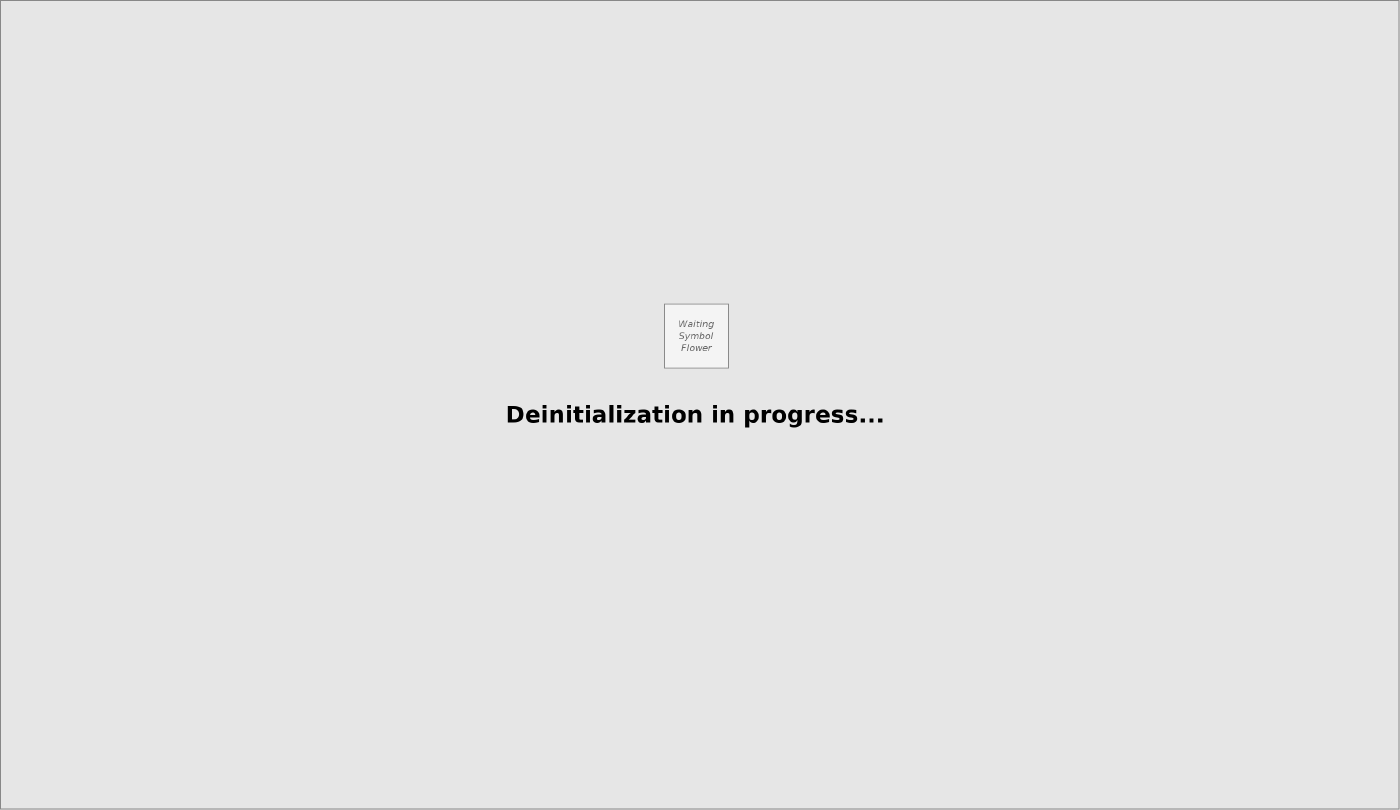
VISUALIZATION PageAborting  // 1520x880
    Group (530,330 450x140)
        WaitingSymbolFlower (191,0 70x70)
        Label (0,100 450x40), "Deinitialization in progress..."
END_VISUALIZATION

// ---- VISUs/Pages/PageAlarms.TcVIS
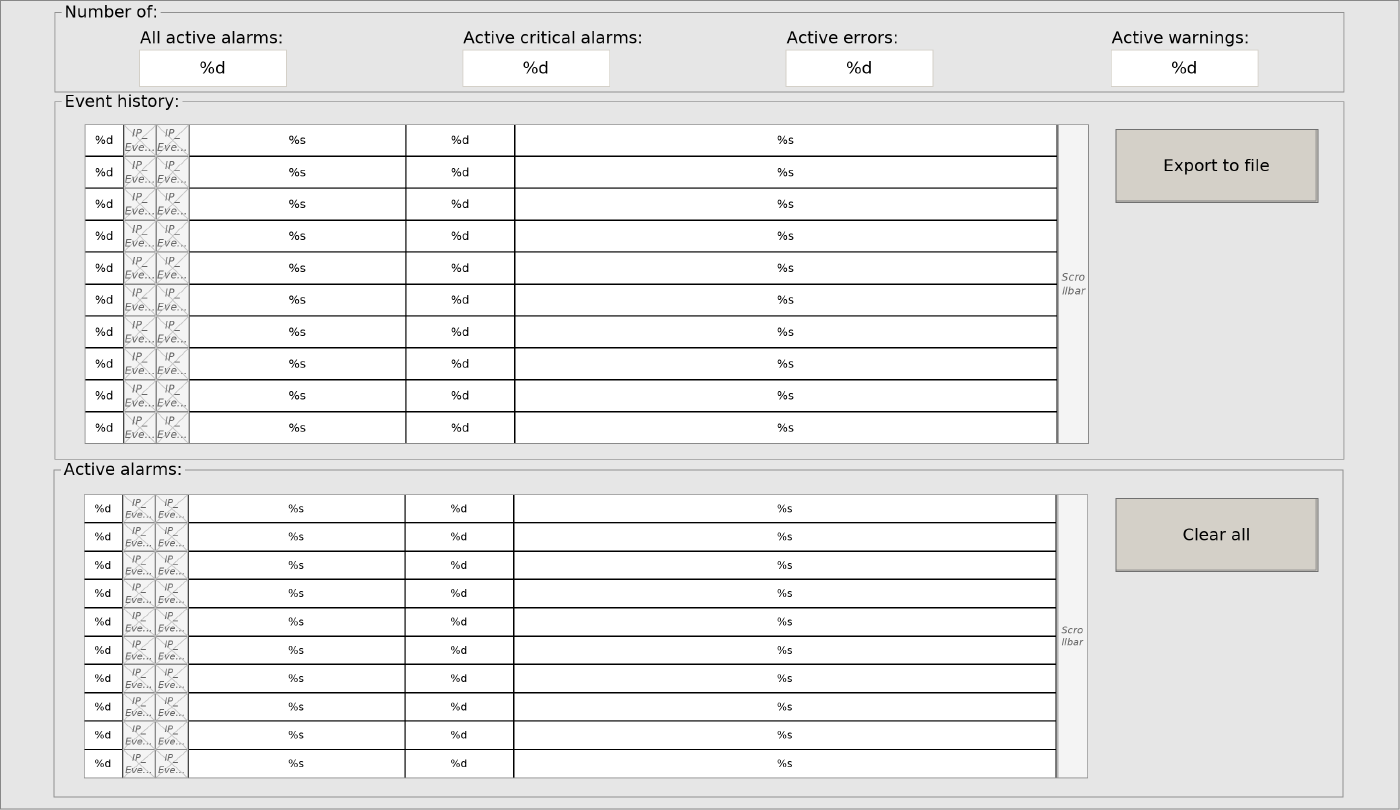
VISUALIZATION PageAlarms  // 1520x880
VAR_IN_OUT
	btnClearAllAlarms 	: BOOL;
	btnExportEvents		: BOOL;
	iActiveAlarms		: UDINT;
	iActiveCritical		: UDINT;
	iActiveErrors		: UDINT;
	iActiveWarrnings	: UDINT;
	arrEvents			: ARRAY[1..PSE_UniversalBlocks.iMAX_EVENTS] OF ST_Event;
	arrAlarms			: ARRAY[1..PSE_UniversalBlocks.iMAX_EVENTS] OF ST_Event;
END_VAR
    GroupBox (58,502 1400x364), "Active alarms:"
        Frame (33,35 1090x308)
            shows EventTable(data := arrAlarms)
        Button (1153,39 220x80), "Clear all"
            tap btnClearAllAlarms
    GroupBox (59,5 1400x95), "Number of:"
        Label (90,21 210x30), "All active alarms:"
        Textfield (92,49 160x40), "%d", text variable: iActiveAlarms, text list: ''
        Label (441,21 234x30), "Active critical alarms:"
        Textfield (443,49 160x40), "%d", text variable: iActiveCritical, text list: ''
        Label (792,21 210x30), "Active errors:"
        Label (1145,21 210x30), "Active warnings:"
        Textfield (794,49 160x40), "%d", text variable: iActiveErrors, text list: ''
        Textfield (1147,49 160x40), "%d", text variable: iActiveWarrnings, text list: ''
    GroupBox (59,102 1400x397), "Event history:"
        Frame (33,33 1090x347)
            shows EventTable(data := arrEvents)
        Button (1152,38 220x80), "Export to file"
            tap btnExportEvents
END_VISUALIZATION

// ---- VISUs/Pages/PageManualCylinders.TcVIS
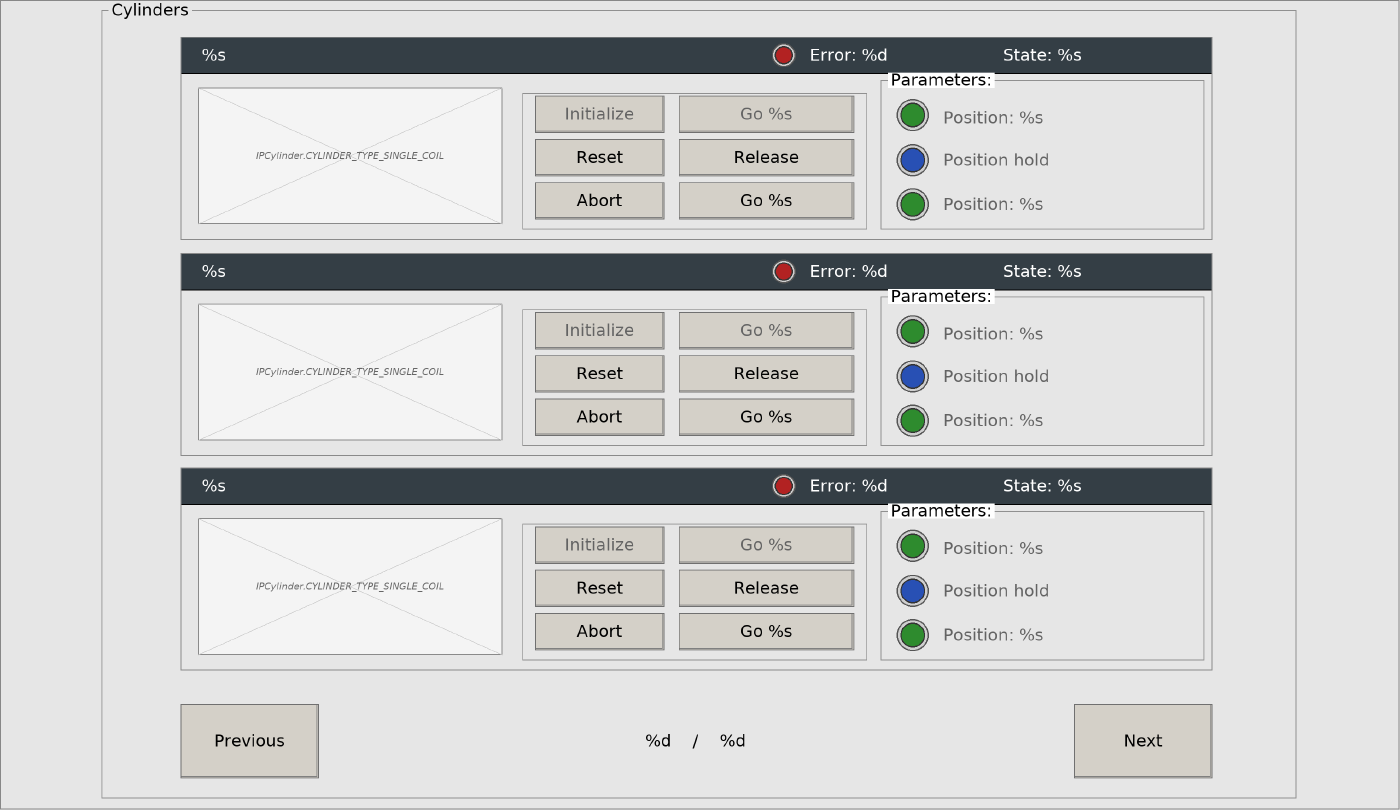
VISUALIZATION PageManualCylinders  // 1520x880
VAR_IN_OUT
	btnPrevious			: BOOL;
	btnNext				: BOOL;
	bPreviousInvisible	: BOOL;
	bNextInvisible		: BOOL;
	stCylinderEmpty		: ARRAY[1..3] OF BOOL;
	stCyliner			: ARRAY[1..3] OF ST_VisuCtrlCylinderFrame;
	iCylinderSelectedPageIndex	: USINT;
	iCylinderTotalPageIndex 	: USINT;
END_VAR
    GroupBox (110,3 1297x864), "Cylinders"
        Button (86,762 150x80), "Previous", invisible if: bPreviousInvisible
            tap btnPrevious
        Button (1056,762 150x80), "Next", invisible if: bNextInvisible
            tap btnNext
        Frame (86,37 1120x220), invisible if: stCylinderEmpty[1]
            shows SingleCylinder(stCylinder := stCyliner[1])
        Frame (86,272 1120x220), invisible if: stCylinderEmpty[2]
            shows SingleCylinder(stCylinder := stCyliner[2])
        Frame (86,505 1120x220), invisible if: stCylinderEmpty[3]
            shows SingleCylinder(stCylinder := stCyliner[3])
        Rectangle (580,777 130x50), "/"
        Rectangle (580,777 50x50), "%d", text variable: iCylinderSelectedPageIndex+1
        Rectangle (661,777 50x50), "%d", text variable: iCylinderTotalPageIndex+1
END_VISUALIZATION

// ---- VISUs/Pages/PageManualRobots.TcVIS
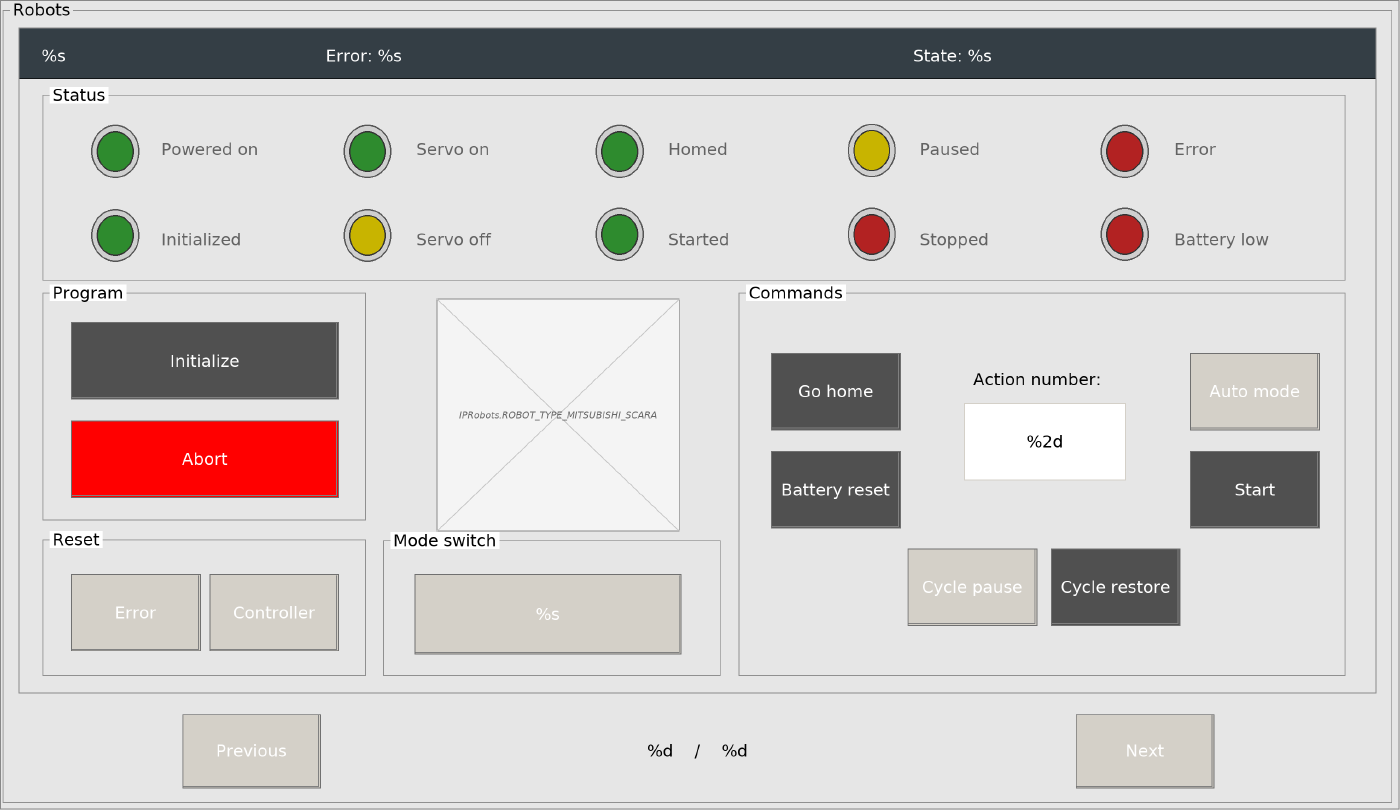
VISUALIZATION PageManualRobots  // 1520x880
VAR_IN_OUT
	btnPrevious			: BOOL;
	btnNext				: BOOL;
	bPreviousInvisible	: BOOL;
	bNextInvisible		: BOOL;
	stRobotEmpty		: ARRAY[1..1] OF BOOL;
	stRobot				: ARRAY[1..1] OF ST_VisuCtrlRobotFrame;
	iRobotSelectedPageIndex	: USINT;
	iRobotTotalPageIndex 	: USINT;
	
END_VAR
    GroupBox (3,3 1508x869), "Robots"
        Button (195,773 150x80), "Previous", invisible if: bPreviousInvisible
            tap btnPrevious
        Button (1165,773 150x80), "Next", invisible if: bNextInvisible
            tap btnNext
        Frame (17,27 1474x723), invisible if: stRobotEmpty[1]
            shows SingleRobot(stRobot := stRobot[1])
        Rectangle (689,788 130x50), "/"
        Rectangle (689,788 50x50), "%d", text variable: iRobotSelectedPageIndex+1
        Rectangle (770,788 50x50), "%d", text variable: iRobotTotalPageIndex+1
END_VISUALIZATION

// ---- VISUs/Pages/PageManualInputs.TcVIS
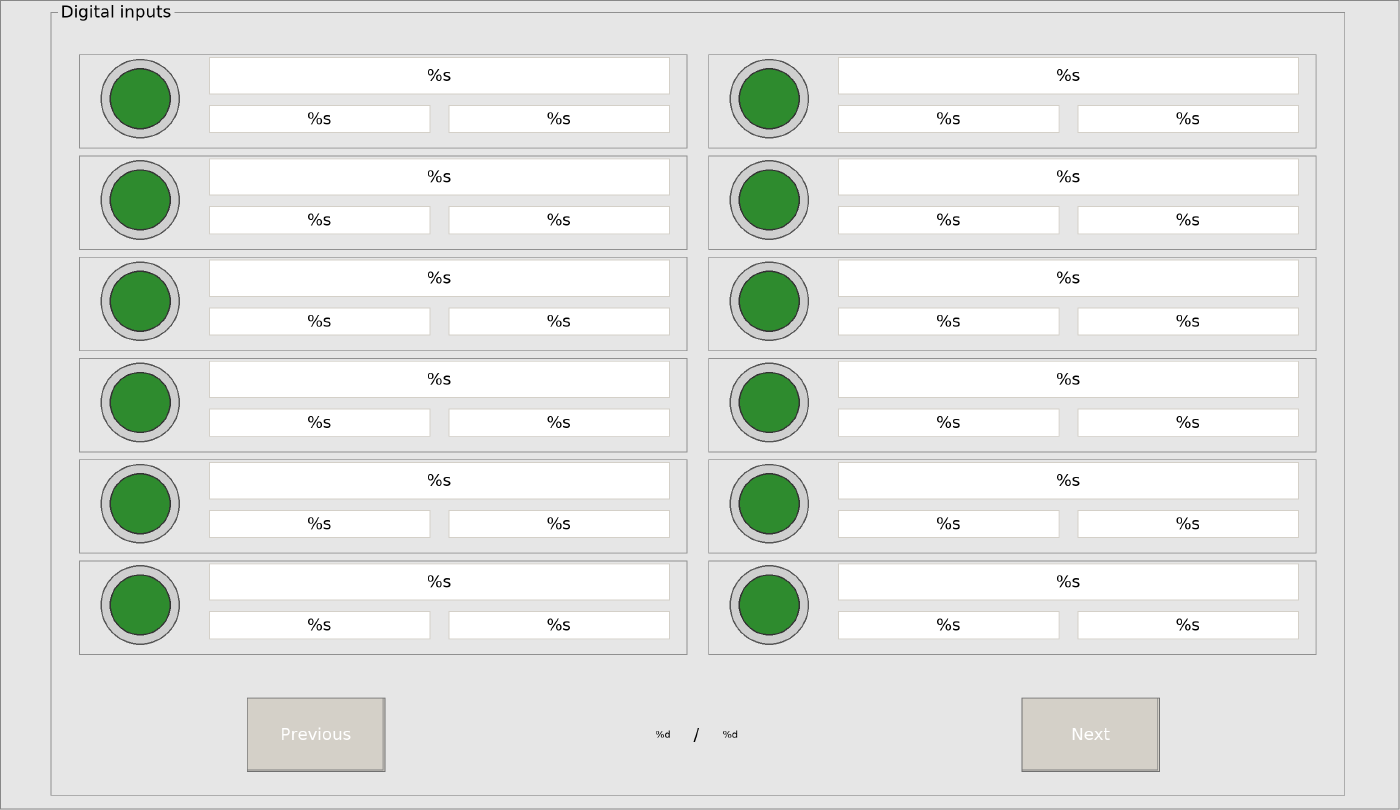
VISUALIZATION PageManualInputs  // 1520x880
VAR_IN_OUT
	btnPrevious			: BOOL;
	btnNext				: BOOL;
	
	bPreviousInvisible	: BOOL;
	bNextInvisible		: BOOL;
	
	stDigitalInputEmpty	: ARRAY[1..12] OF BOOL;
	stDigitalInputData	: ARRAY[1..12] OF ST_VisuCtrlInputFrame;
	
	iInputSelectedPageIndex		: USINT;
	iInputTotalPageIndex 		: USINT;
END_VAR
    GroupBox (55,5 1405x859), "Digital inputs"
        Rectangle (713,768 50x50), "%d", text variable: iInputTotalPageIndex+1
        Rectangle (640,768 50x50), "%d", text variable: iInputSelectedPageIndex+1
        Rectangle (636,768 130x50), "/"
        Button (213,753 150x80), "Previous", invisible if: bPreviousInvisible
            tap btnPrevious
        Button (1054,753 150x80), "Next", invisible if: bNextInvisible
            tap btnNext
        Frame (31,46 660x110), invisible if: stDigitalInputEmpty[1]
            shows SingleDigitalInput(stDigitalInput := stDigitalInputData[1])
        Frame (31,156 660x110), invisible if: stDigitalInputEmpty[2]
            shows SingleDigitalInput(stDigitalInput := stDigitalInputData[2])
        Frame (31,266 660x110), invisible if: stDigitalInputEmpty[3]
            shows SingleDigitalInput(stDigitalInput := stDigitalInputData[3])
        Frame (31,376 660x110), invisible if: stDigitalInputEmpty[4]
            shows SingleDigitalInput(stDigitalInput := stDigitalInputData[4])
        Frame (31,486 660x110), invisible if: stDigitalInputEmpty[5]
            shows SingleDigitalInput(stDigitalInput := stDigitalInputData[5])
        Frame (31,596 660x110), invisible if: stDigitalInputEmpty[6]
            shows SingleDigitalInput(stDigitalInput := stDigitalInputData[6])
        Frame (714,46 660x110), invisible if: stDigitalInputEmpty[7]
            shows SingleDigitalInput(stDigitalInput := stDigitalInputData[7])
    Frame (769,161 660x110), invisible if: stDigitalInputEmpty[8]
        shows SingleDigitalInput(stDigitalInput := stDigitalInputData[8])
    Frame (769,271 660x110), invisible if: stDigitalInputEmpty[9]
        shows SingleDigitalInput(stDigitalInput := stDigitalInputData[9])
    Frame (769,381 660x110), invisible if: stDigitalInputEmpty[10]
        shows SingleDigitalInput(stDigitalInput := stDigitalInputData[10])
    Frame (769,491 660x110), invisible if: stDigitalInputEmpty[11]
        shows SingleDigitalInput(stDigitalInput := stDigitalInputData[11])
    Frame (769,601 660x110), invisible if: stDigitalInputEmpty[12]
        shows SingleDigitalInput(stDigitalInput := stDigitalInputData[12])
END_VISUALIZATION

// ---- VISUs/Pages/PageManualAxis.TcVIS
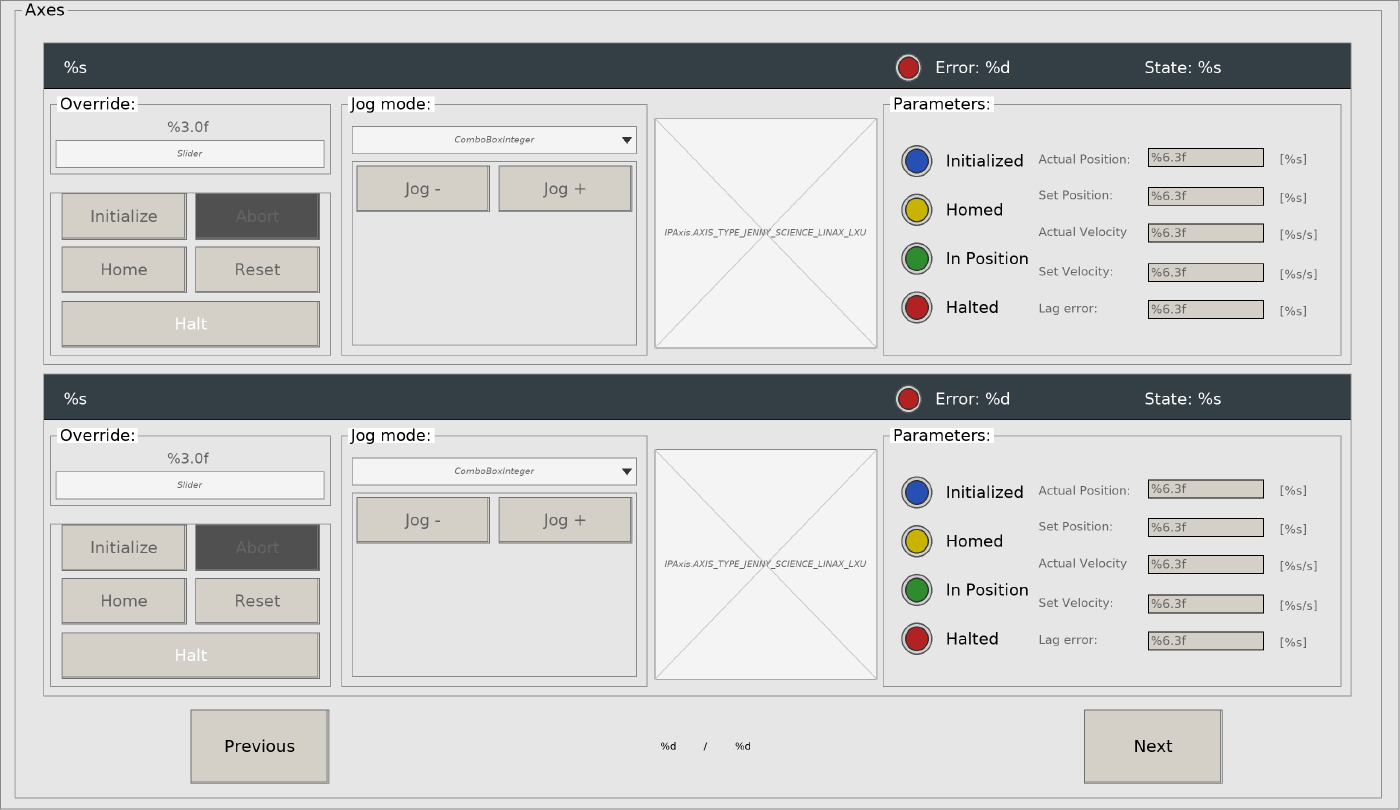
VISUALIZATION PageManualAxis  // 1520x880
VAR_IN_OUT
	btnPrevious			: BOOL;
	btnNext				: BOOL;
	bPreviousInvisible	: BOOL;
	bNextInvisible		: BOOL;
	stAxisEmpty			: ARRAY[0..1] OF BOOL;
	stAxis				: ARRAY[0..1] OF ST_VisuCtrlAxisFrame;
	iAxisSelectedPageIndex		: USINT;
	iAxisTotalPageIndex 		: USINT;
END_VAR
    GroupBox (16,3 1484x864), "Axes"
        Frame (31,43 1420x350), invisible if: stAxisEmpty[0]
            shows SingleAxis(stAxis := stAxis[0])
        Button (1161,768 150x80), "Next", invisible if: bNextInvisible
            tap btnNext
        Button (191,768 150x80), "Previous", invisible if: bPreviousInvisible
            tap btnPrevious
        Frame (31,403 1420x350), invisible if: stAxisEmpty[1]
            shows SingleAxis(stAxis := stAxis[1])
        Rectangle (685,783 130x50), "/"
        Rectangle (685,783 50x50), "%d", text variable: iAxisSelectedPageIndex+1
        Rectangle (766,783 50x50), "%d", text variable: iAxisTotalPageIndex+1
END_VISUALIZATION

// ---- VISUs/Pages/PageManualOutputs.TcVIS
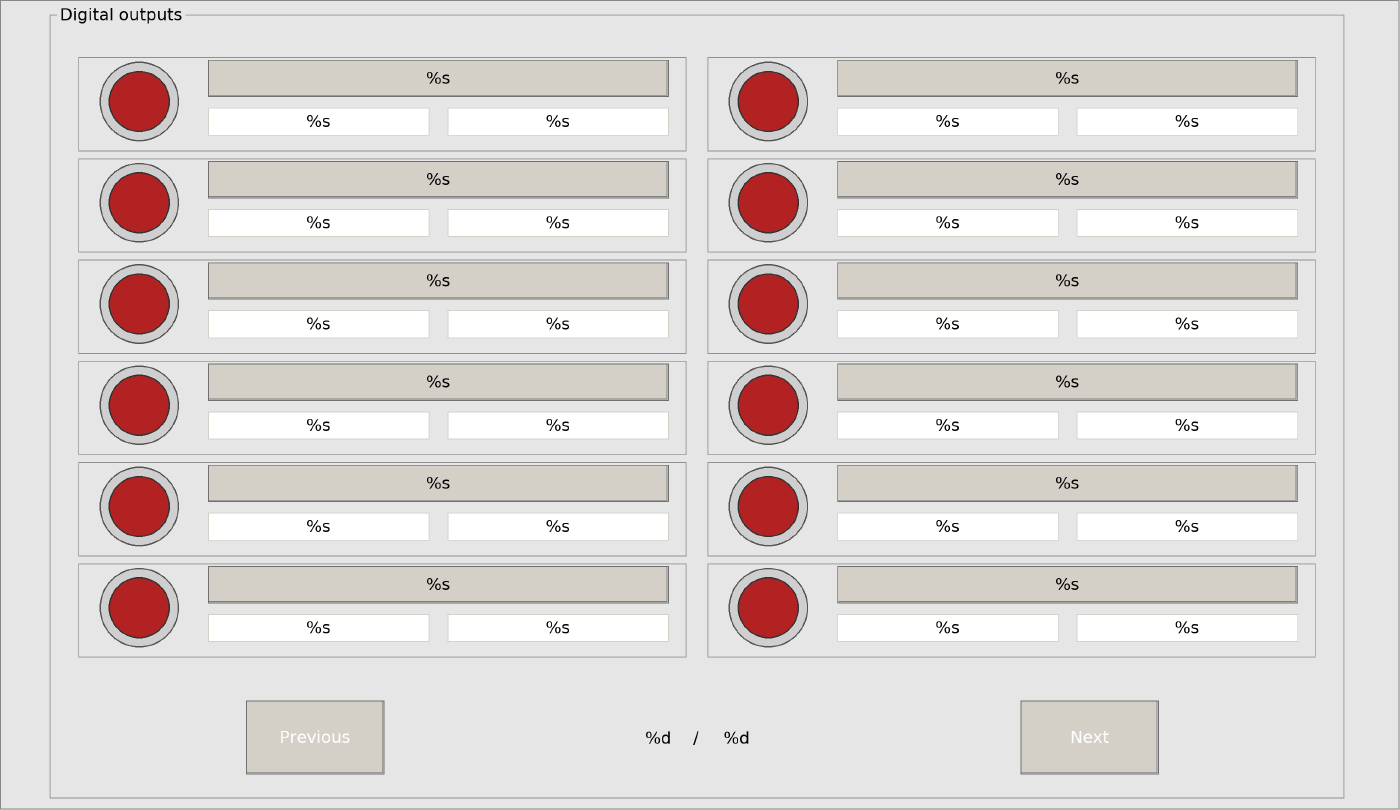
VISUALIZATION PageManualOutputs  // 1520x880
VAR_IN_OUT
	btnPrevious			: BOOL;
	btnNext				: BOOL;
	
	bPreviousInvisible	: BOOL;
	bNextInvisible		: BOOL;
	
	stDigitalOutputEmpty: ARRAY[1..12] OF BOOL;
	stDigitalOutputData	: ARRAY[1..12] OF ST_VisuCtrlOutputFrame;
	
	iOutputSelectedPageIndex	: USINT;
	iOutputTotalPageIndex 		: USINT;
END_VAR
    GroupBox (54,8 1405x859), "Digital outputs"
        Rectangle (721,769 50x50), "%d", text variable: iOutputTotalPageIndex + 1
        Rectangle (636,769 50x50), "%d", text variable: iOutputSelectedPageIndex+1
        Rectangle (636,768 131x51), "/"
        Button (213,753 150x80), "Previous", invisible if: bPreviousInvisible
            tap btnPrevious
        Button (1054,753 150x80), "Next", invisible if: bNextInvisible
            tap btnNext
        Frame (31,46 660x110), invisible if: stDigitalOutputEmpty[1]
            shows SingleDigitalOutput(stDigitalOutput := stDigitalOutputData[1])
        Frame (31,156 660x110), invisible if: stDigitalOutputEmpty[2]
            shows SingleDigitalOutput(stDigitalOutput := stDigitalOutputData[2])
        Frame (31,266 660x110), invisible if: stDigitalOutputEmpty[3]
            shows SingleDigitalOutput(stDigitalOutput := stDigitalOutputData[3])
        Frame (31,376 660x110), invisible if: stDigitalOutputEmpty[4]
            shows SingleDigitalOutput(stDigitalOutput := stDigitalOutputData[4])
        Frame (31,486 660x110), invisible if: stDigitalOutputEmpty[5]
            shows SingleDigitalOutput(stDigitalOutput := stDigitalOutputData[5])
        Frame (31,596 660x110), invisible if: stDigitalOutputEmpty[6]
            shows SingleDigitalOutput(stDigitalOutput := stDigitalOutputData[6])
        Frame (714,46 660x110), invisible if: stDigitalOutputEmpty[7]
            shows SingleDigitalOutput(stDigitalOutput := stDigitalOutputData[7])
    Frame (768,164 660x110), invisible if: stDigitalOutputEmpty[8]
        shows SingleDigitalOutput(stDigitalOutput := stDigitalOutputData[8])
    Frame (768,274 660x110), invisible if: stDigitalOutputEmpty[9]
        shows SingleDigitalOutput(stDigitalOutput := stDigitalOutputData[9])
    Frame (768,384 660x110), invisible if: stDigitalOutputEmpty[10]
        shows SingleDigitalOutput(stDigitalOutput := stDigitalOutputData[10])
    Frame (768,494 660x110), invisible if: stDigitalOutputEmpty[11]
        shows SingleDigitalOutput(stDigitalOutput := stDigitalOutputData[11])
    Frame (768,604 660x110), invisible if: stDigitalOutputEmpty[12]
        shows SingleDigitalOutput(stDigitalOutput := stDigitalOutputData[12])
END_VISUALIZATION

// ---- VISUs/Pages/PageManualSafety.TcVIS
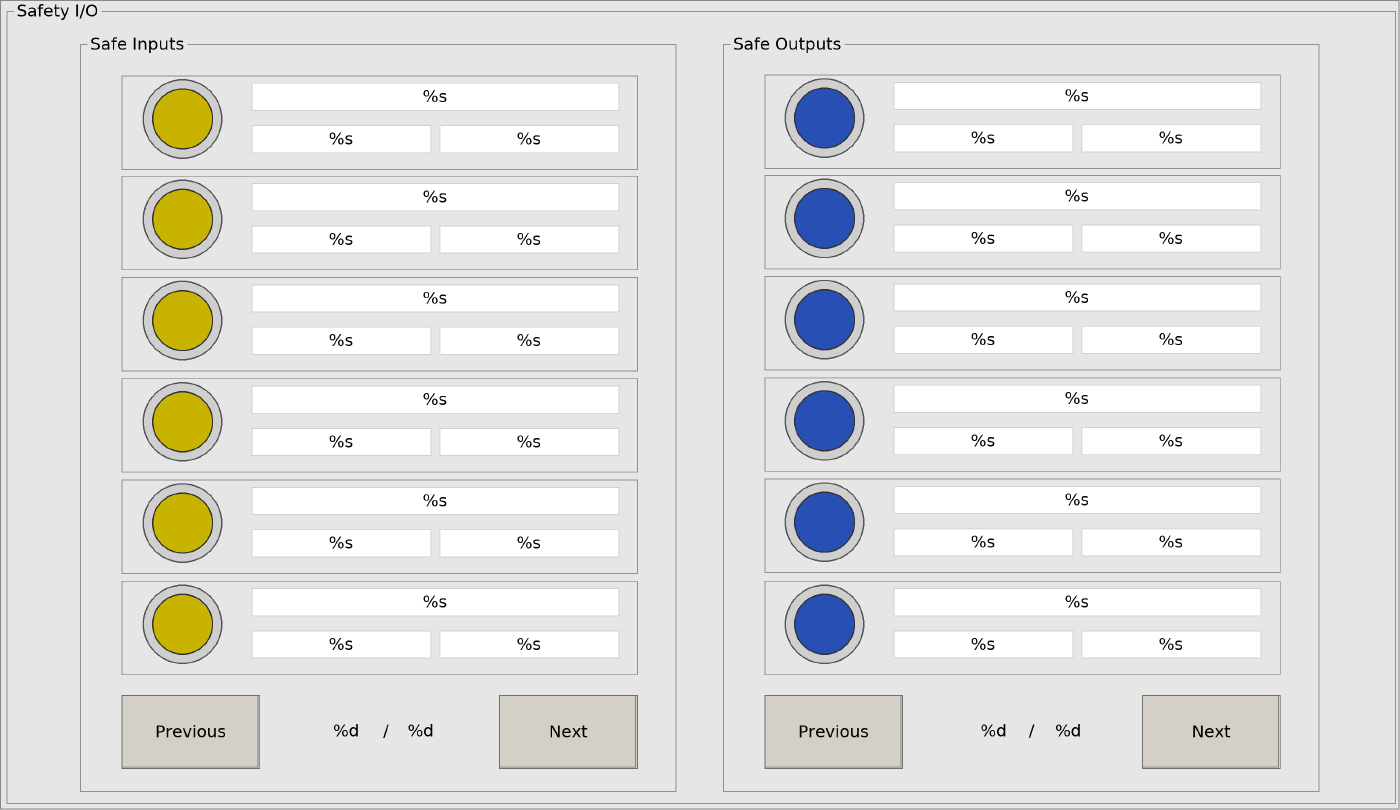
VISUALIZATION PageManualSafety  // 1520x880
VAR_IN_OUT
	btnNextInput			: BOOL;				(*  *)
	btnPreviousInput		: BOOL;				(*  *)
	btnNextOutput			: BOOL;				(*  *)
	btnPreviousOutput		: BOOL;				(*  *)
	
	bNextInvisibleInput		: BOOL;				(*  *)
	bPreviousInvisibleInput	: BOOL;				(*  *)
	bNextInvisibleOutput	: BOOL;				(*  *)
	bPreviousInvisibleOutput: BOOL;				(*  *)	
	
	iSafeInputSelectedPageIndex		: USINT;
	iSafeInputTotalPageIndex 		: USINT;
	iSafeOutputSelectedPageIndex	: USINT;
	iSafeOutputTotalPageIndex 		: USINT;
	
	stSafeOutputEmpty		: ARRAY[1..6] OF BOOL;
	stSafeOutputData		: ARRAY[1..6] OF ST_VisuCtrlOutputFrame;
	stSafeInputEmpty		: ARRAY[1..6] OF BOOL;
	stSafeInputData			: ARRAY[1..6] OF ST_VisuCtrlInputFrame;
END_VAR
    GroupBox (7,4 1508x869), "Safety I/O"
        GroupBox (80,36 647x820), "Safe Inputs"
            Frame (45,583 560x110), invisible if: stSafeInputEmpty[6]
                shows SingleSafeInput(stDigitalInput := stSafeInputData[6])
            Rectangle (345,729 50x50), "%d", text variable: iSafeInputTotalPageIndex+1
            Rectangle (264,729 50x50), "%d", text variable: iSafeInputSelectedPageIndex+1
            Rectangle (1461,1588 130x50), "/"
            Button (45,715 150x80), "Previous", pressed state: btnPreviousInput, invisible if: bPreviousInvisibleInput
                tap btnPreviousInput
            Button (455,715 150x80), "Next", pressed state: btnNextInput, invisible if: bNextInvisibleInput
                tap btnNextInput
            Frame (45,473 560x110), invisible if: stSafeInputEmpty[5]
                shows SingleSafeInput(stDigitalInput := stSafeInputData[5])
            Frame (45,363 560x110), invisible if: stSafeInputEmpty[4]
                shows SingleSafeInput(stDigitalInput := stSafeInputData[4])
            Frame (45,253 560x110), invisible if: stSafeInputEmpty[3]
                shows SingleSafeInput(stDigitalInput := stSafeInputData[3])
            Frame (45,143 560x110), invisible if: stSafeInputEmpty[2]
                shows SingleSafeInput(stDigitalInput := stSafeInputData[2])
            Frame (45,34 560x110), invisible if: stSafeInputEmpty[1]
                shows SingleSafeInput(stDigitalInput := stSafeInputData[1])
            Rectangle (267,729 130x50), "/"
        GroupBox (778,36 647x820), "Safe Outputs"
            Frame (45,583 560x110), invisible if: stSafeOutputEmpty[6]
                shows SingleSafeOutput(stDigitalOutput := stSafeOutputData[6])
            Rectangle (350,729 50x50), "%d", text variable: iSafeOutputTotalPageIndex+1
            Rectangle (269,729 50x50), "%d", text variable: iSafeOutputSelectedPageIndex+1
            Button (45,715 150x80), "Previous", pressed state: btnPreviousOutput, invisible if: bPreviousInvisibleOutput
                tap btnPreviousOutput
            Button (455,715 150x80), "Next", pressed state: btnNextOutput, invisible if: bNextInvisibleOutput
                tap btnNextOutput
            Frame (45,472 560x110), invisible if: stSafeOutputEmpty[5]
                shows SingleSafeOutput(stDigitalOutput := stSafeOutputData[5])
            Frame (45,362 560x110), invisible if: stSafeOutputEmpty[4]
                shows SingleSafeOutput(stDigitalOutput := stSafeOutputData[4])
            Frame (45,252 560x110), invisible if: stSafeOutputEmpty[3]
                shows SingleSafeOutput(stDigitalOutput := stSafeOutputData[3])
            Frame (45,142 560x110), invisible if: stSafeOutputEmpty[2]
                shows SingleSafeOutput(stDigitalOutput := stSafeOutputData[2])
            Frame (45,33 560x110), invisible if: stSafeOutputEmpty[1]
                shows SingleSafeOutput(stDigitalOutput := stSafeOutputData[1])
            Rectangle (270,729 130x50), "/"
END_VISUALIZATION

// ---- VISUs/Pages/PageReadyInitialized.TcVIS
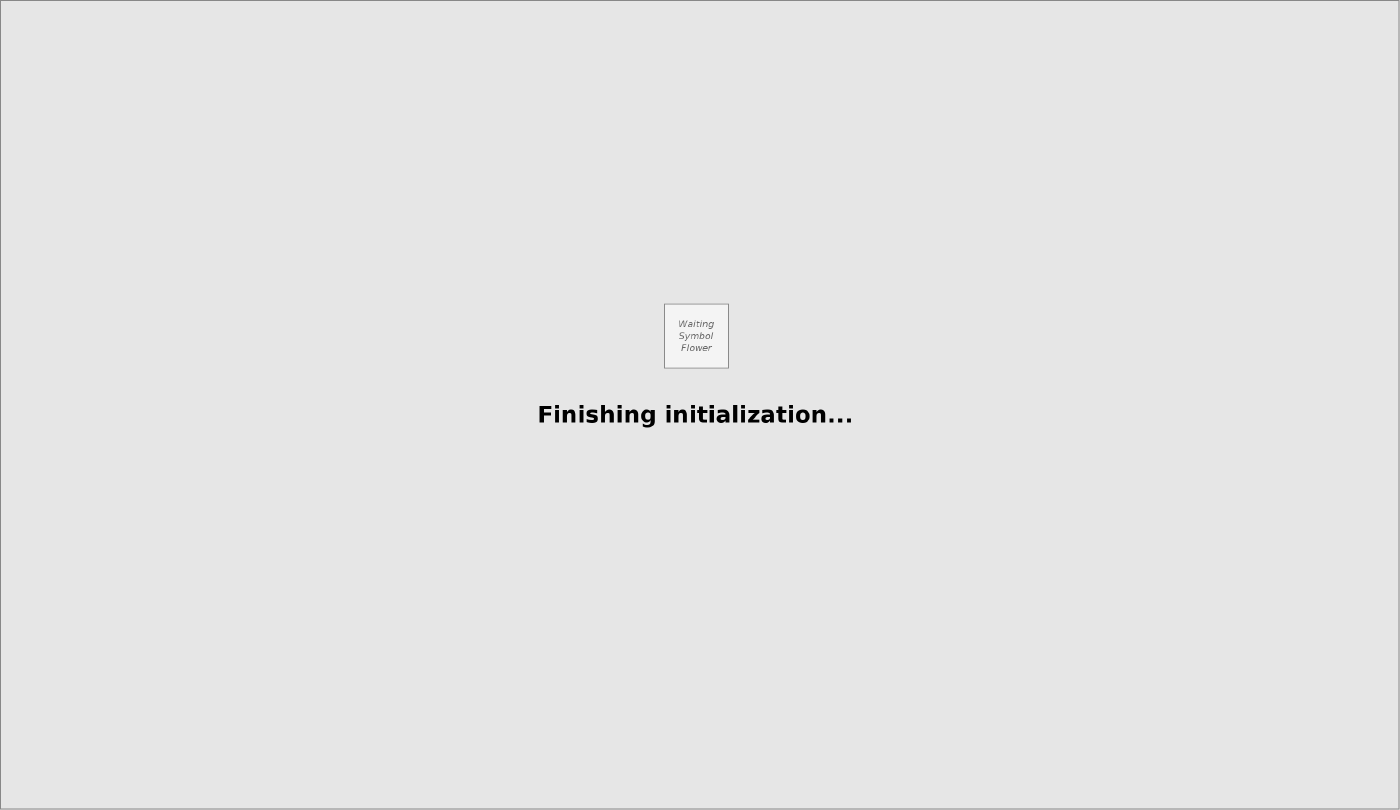
VISUALIZATION PageReadyInitialized  // 1520x880
    WaitingSymbolFlower (721,330 70x70)
    Label (530,430 450x40), "Finishing initialization..."
END_VISUALIZATION

// ---- VISUs/Pages/PageRecipesManager.TcVIS
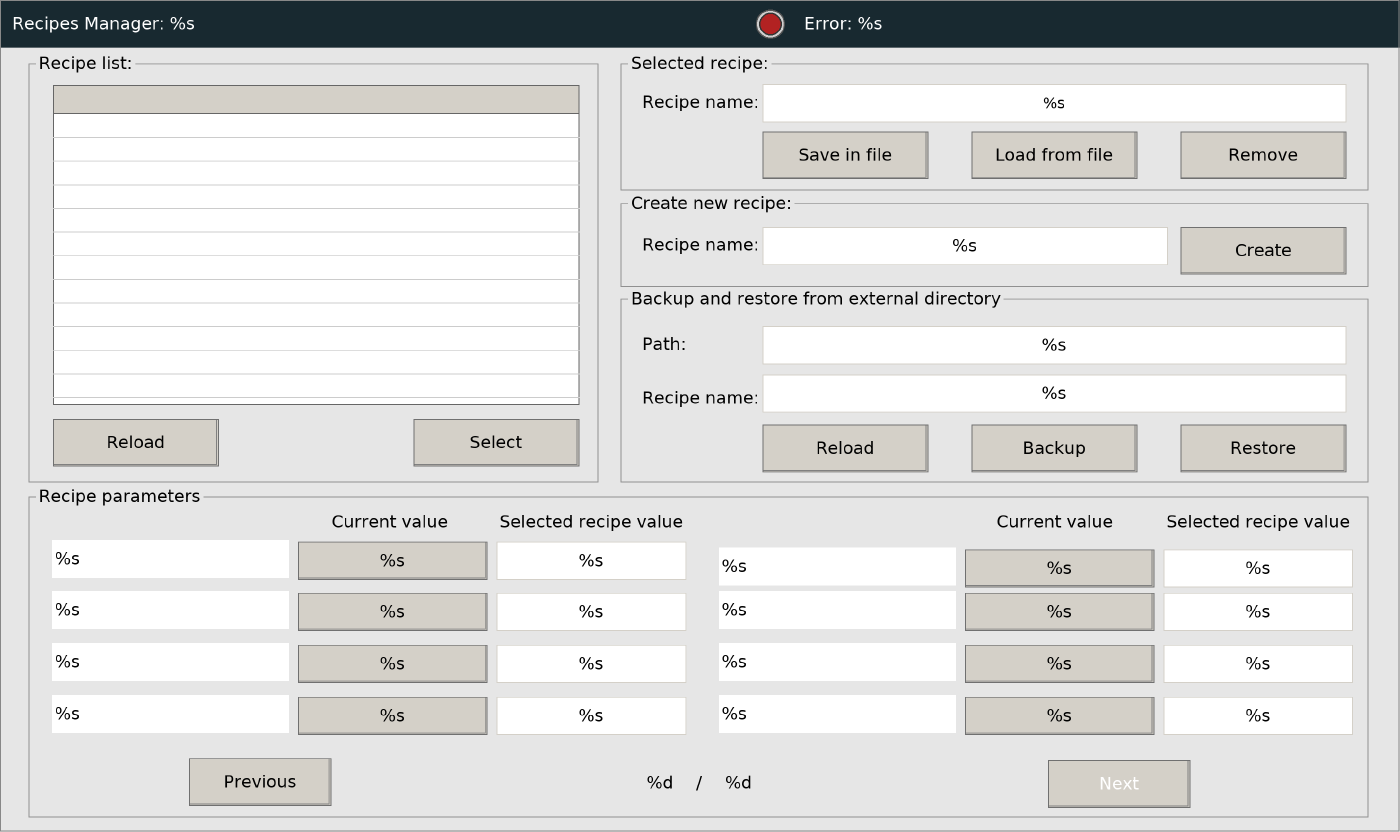
VISUALIZATION PageRecipesManager  // 1480x880
VAR_IN_OUT
	(* Recipe control - buttons *)
	btnCreate						: BOOL;						(* Create recipe button *)
	btnSelect						: BOOL;						(* Select recipe from table button*)
	btnLoad							: BOOL;						(* Load recipe from file button *)
	btnRead							: BOOL;						(* Read recipe to file button *)
	btnReload 						: BOOL;						(* Reload recipes button *)
	btnBackup						: BOOL;						(* Backup recipes to external directory button *)
	btnRestore						: BOOL;						(* Restore recipes from external directory button *)
	btnRecipeNext					: BOOL;						(* Go to next page with recipe parameters *)
	btnRecipePrevious				: BOOL;						(* Go to previous page with recipe parameters *)
	btnRemove						: BOOL;
	btnReloadExternal				: BOOL;
		
	(* Recipe control - visibility *)
	bReloadInvisible				: BOOL;						(* Makes reload button invisible *)
	bRecipeNextInvisible			: BOOL;						(* Makes next button invisible *)
	bRecipePreviousInvisible		: BOOL;						(* Makes previous button invisible *)
	bRecipeCreateInvisible			: BOOL;						(* Makes create group box invisible *)
	bRecipeBackupRestoreInvisible	: BOOL;						(* Makes backup and restore group box invisible *)
	bNoRecipeSelected				: BOOL;
	
	(* Recipe control - control disabled *)
	bRecipeCreateDisabled			: BOOL;						(* Disable access to create recipe group box *)
	bRecipeBackupRestoreDisabled	: BOOL;						(* Disable access to backup and restore group box *)
	
	(* Recipe control - status *)
	bError							: BOOL;						(* Error occured while executing last command *)
	eRecipesManagerReturns			: E_RecipesManagerReturns;	(* Result of last executed command *)
	eReacipeManagerState			: E_RecipesManagerState;	(* Current state of Recipe Manager *)
	
	(* Recipe control - parameters for recipes manager *)
	iSelectedRecipe					: INT;						(* Number of selected row in Available Recipes table *)
	sSelectedRecipe					: STRING;					(* Current selected recipe name - changes affter trigger from btnSelect *)
	sNewRecipeName					: STRING;					(* Name for new recipe *)
	sRestoreBackupPath				: STRING;				(* Path for backup/restoring of recipes *)
	sRestoreBackupRecipeName		: STRING;	
	arrRecipeNames					: ARRAY	[0..127] OF STRING;	(* Names of all detected recipes *)
	
	(* Recipe control - parameters data *)
	arrRecipeParameterFrameEmpty 	: ARRAY [0..7] OF BOOL;								(*  *)
	arrRecipeParameterFrameData		: ARRAY [0..7] OF ST_VisuCtrlRecipeParameter;		(*  *)
	arrRecipeParameterFrameType		: ARRAY [0..7] OF E_VisuCtrlRecipeParameterType;	(*  *)
	
	iRecipeSelectedPageIndex	: USINT;
	iRecipeTotalPageIndex 		: USINT;
END_VAR
    Rectangle (0,0 1480x50)
    Textfield (10,0 350x50), "Recipes Manager: %s", text list: 'TL_RecipesManagerStatus', text index: eReacipeManagerState
    GroupBox (30,517 1416x347), "Recipe parameters"
        Label (312,20 140x30), "Current value"
        Label (490,20 210x30), "Selected recipe value"
        Label (1010,20 150x30), "Current value"
        Label (1195,20 210x30), "Selected recipe value"
        Button (170,285 150x50), "Previous", invisible if: bRecipePreviousInvisible
            tap btnRecipePrevious
        Button (1078,287 150x50), "Next", invisible if: bRecipeNextInvisible
            tap btnRecipeNext
        Rectangle (644,286 130x50), "/"
        Rectangle (643,286 50x50), "%d", text variable: iRecipeSelectedPageIndex+1
        Rectangle (726,286 50x50), "%d", text variable: iRecipeTotalPageIndex+1
        Frame (20,100 680x60), invisible if: arrRecipeParameterFrameEmpty[1], frame switch variable: arrRecipeParameterFrameType[1]
            shows SingleRecipesParameterTypeBool(stRecipeParameter := arrRecipeParameterFrameData[1])
            shows SingleRecipesParameterTypeInteger(stRecipeParameter := arrRecipeParameterFrameData[1])
            shows SingleRecipesParameterTypeReal(stRecipeParameter := arrRecipeParameterFrameData[1])
            shows SingleRecipesParameterTypeString(stRecipeParameter := arrRecipeParameterFrameData[1])
        Frame (20,155 680x60), invisible if: arrRecipeParameterFrameEmpty[2], frame switch variable: arrRecipeParameterFrameType[2]
            shows SingleRecipesParameterTypeBool(stRecipeParameter := arrRecipeParameterFrameData[2])
            shows SingleRecipesParameterTypeInteger(stRecipeParameter := arrRecipeParameterFrameData[2])
            shows SingleRecipesParameterTypeReal(stRecipeParameter := arrRecipeParameterFrameData[2])
            shows SingleRecipesParameterTypeString(stRecipeParameter := arrRecipeParameterFrameData[2])
        Frame (20,210 680x60), invisible if: arrRecipeParameterFrameEmpty[3], frame switch variable: arrRecipeParameterFrameType[3]
            shows SingleRecipesParameterTypeBool(stRecipeParameter := arrRecipeParameterFrameData[3])
            shows SingleRecipesParameterTypeInteger(stRecipeParameter := arrRecipeParameterFrameData[3])
            shows SingleRecipesParameterTypeReal(stRecipeParameter := arrRecipeParameterFrameData[3])
            shows SingleRecipesParameterTypeString(stRecipeParameter := arrRecipeParameterFrameData[3])
        Frame (725,54 680x60), invisible if: arrRecipeParameterFrameEmpty[4], frame switch variable: arrRecipeParameterFrameType[4]
            shows SingleRecipesParameterTypeBool(stRecipeParameter := arrRecipeParameterFrameData[4])
            shows SingleRecipesParameterTypeInteger(stRecipeParameter := arrRecipeParameterFrameData[4])
            shows SingleRecipesParameterTypeReal(stRecipeParameter := arrRecipeParameterFrameData[4])
            shows SingleRecipesParameterTypeString(stRecipeParameter := arrRecipeParameterFrameData[4])
        Frame (725,100 680x60), invisible if: arrRecipeParameterFrameEmpty[5], frame switch variable: arrRecipeParameterFrameType[5]
            shows SingleRecipesParameterTypeBool(stRecipeParameter := arrRecipeParameterFrameData[5])
            shows SingleRecipesParameterTypeInteger(stRecipeParameter := arrRecipeParameterFrameData[5])
            shows SingleRecipesParameterTypeReal(stRecipeParameter := arrRecipeParameterFrameData[5])
            shows SingleRecipesParameterTypeString(stRecipeParameter := arrRecipeParameterFrameData[5])
        Frame (725,155 680x60), invisible if: arrRecipeParameterFrameEmpty[6], frame switch variable: arrRecipeParameterFrameType[6]
            shows SingleRecipesParameterTypeBool(stRecipeParameter := arrRecipeParameterFrameData[6])
            shows SingleRecipesParameterTypeInteger(stRecipeParameter := arrRecipeParameterFrameData[6])
            shows SingleRecipesParameterTypeReal(stRecipeParameter := arrRecipeParameterFrameData[6])
            shows SingleRecipesParameterTypeString(stRecipeParameter := arrRecipeParameterFrameData[6])
        Frame (725,210 680x60), invisible if: arrRecipeParameterFrameEmpty[7], frame switch variable: arrRecipeParameterFrameType[7]
            shows SingleRecipesParameterTypeBool(stRecipeParameter := arrRecipeParameterFrameData[7])
            shows SingleRecipesParameterTypeInteger(stRecipeParameter := arrRecipeParameterFrameData[7])
            shows SingleRecipesParameterTypeReal(stRecipeParameter := arrRecipeParameterFrameData[7])
            shows SingleRecipesParameterTypeString(stRecipeParameter := arrRecipeParameterFrameData[7])
        Frame (20,46 680x60), invisible if: arrRecipeParameterFrameEmpty[0], frame switch variable: arrRecipeParameterFrameType[0]
            shows SingleRecipesParameterTypeBool(stRecipeParameter := arrRecipeParameterFrameData[0])
            shows SingleRecipesParameterTypeInteger(stRecipeParameter := arrRecipeParameterFrameData[0])
            shows SingleRecipesParameterTypeReal(stRecipeParameter := arrRecipeParameterFrameData[0])
            shows SingleRecipesParameterTypeString(stRecipeParameter := arrRecipeParameterFrameData[0])
    GroupBox (30,59 602x451), "Recipe list:", invisible if: bRecipeCreateInvisible, input disabled if: bRecipeCreateDisabled
        Button (26,384 175x50), "Reload", invisible if: bReloadInvisible
            tap btnReload
        Table (26,31 556x338), text list: '', data array: arrRecipeNames
            p1137915858: iSelectedRecipe
            p3854506369: arrRecipeNames[INDEX]
            p2232123230: Available Recipes
        Button (407,384 175x50), "Select"
            tap btnSelect
    GroupBox (656,308 790x202), "Backup and restore from external directory"
        Button (371,141 175x50), "Backup"
            tap btnBackup
        Button (592,141 175x50), "Restore"
            tap btnRestore
        Textfield (150,37 617x40), "%s", text variable: sRestoreBackupPath
            OnMouseClick: write the text variable via VisuDialogs.Keypad
        Label (20,41 150x30), "Path:"
        Textfield (150,88 617x40), "%s", text variable: sRestoreBackupRecipeName
            OnMouseClick: write the text variable via VisuDialogs.Keypad
        Button (150,141 175x50), "Reload"
            tap btnReloadExternal
        Label (20,98 123x30), "Recipe name:"
    GroupBox (656,207 790x96), "Create new recipe:", invisible if: bRecipeCreateInvisible, input disabled if: bRecipeCreateDisabled
        Button (592,33 175x50), "Create"
            tap btnCreate
        Textfield (150,33 428x40), "%s", text variable: sNewRecipeName
            OnMouseClick: write the text variable via VisuDialogs.Keypad
        Label (20,37 150x30), "Recipe name:"
    GroupBox (656,59 790x142), "Selected recipe:", input disabled if: bNoRecipeSelected
        Button (150,80 175x50), "Save in file"
            tap btnRead
        Button (592,80 175x50), "Remove"
            tap btnRemove
        Textfield (150,30 617x40), "%s", text variable: sSelectedRecipe
        Button (371,80 175x50), "Load from file"
            tap btnLoad
        Label (20,34 150x30), "Recipe name:"
    Textfield (847,0 594x50), "Error: %s", text list: 'TL_RecipesManagerReturns', text index: eRecipesManagerReturns
    Lamp1 (797,8 35x35), variable: bError, style: Lamp-Lamp1-Red
END_VISUALIZATION

// ---- VISUs/Pages/PageReset.TcVIS
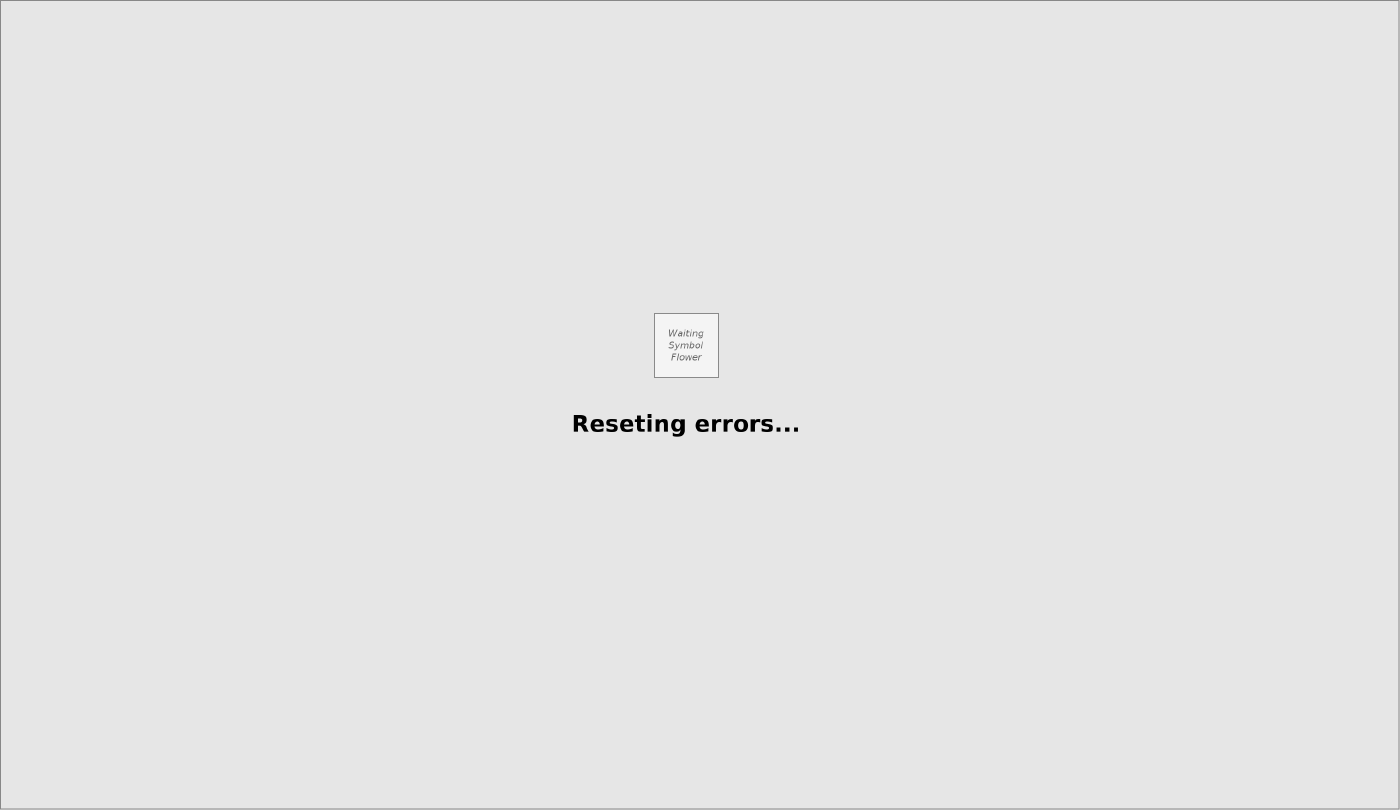
VISUALIZATION PageReset  // 1520x880
    WaitingSymbolFlower (710,340 70x70)
    Label (570,440 350x40), "Reseting errors..."
END_VISUALIZATION

// ---- VISUs/Pages/PageSwitchMode.TcVIS
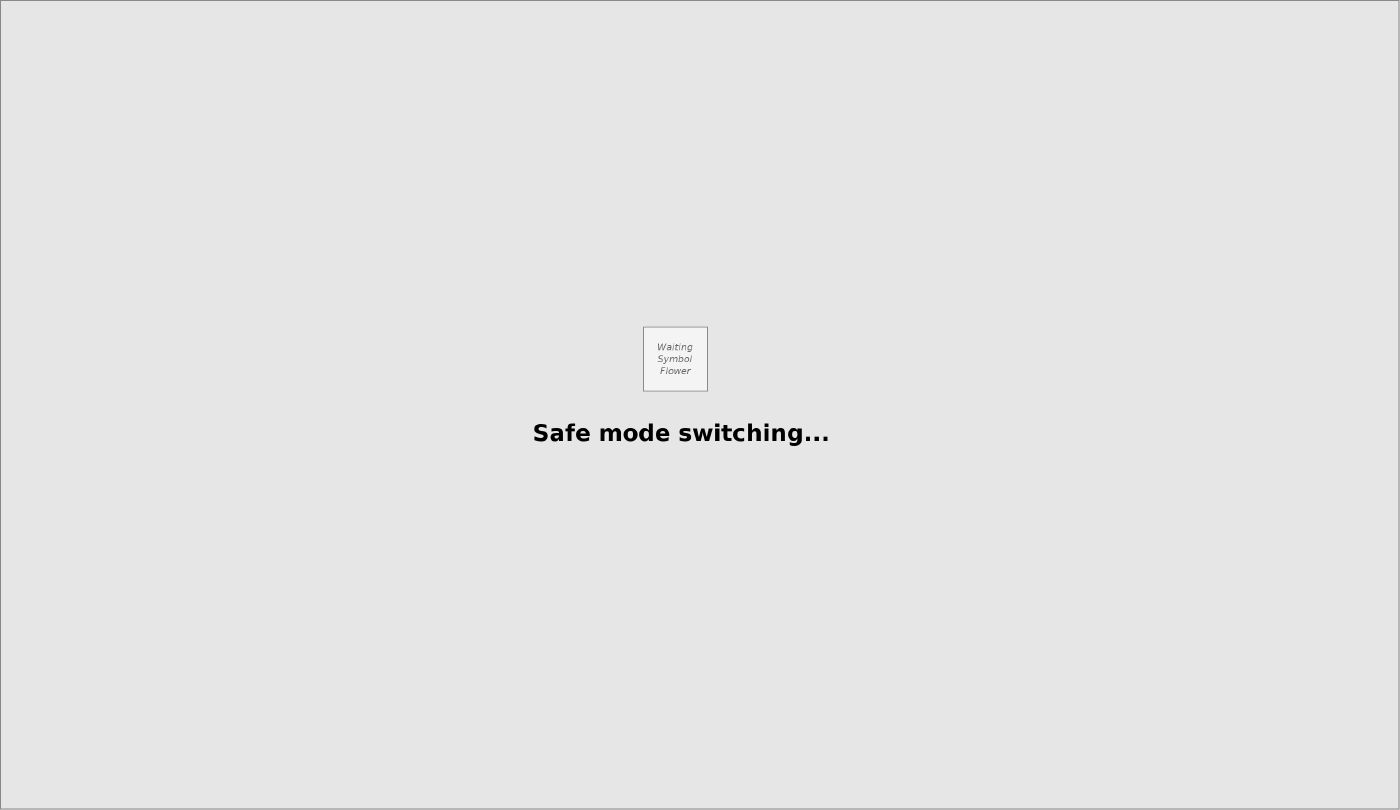
VISUALIZATION PageSwitchMode  // 1520x880
    Label (490,450 500x40), "Safe mode switching..."
    WaitingSymbolFlower (698,355 70x70)
END_VISUALIZATION

// ---- VISUs/Pages/PageXtsDiagnostic.TcVIS
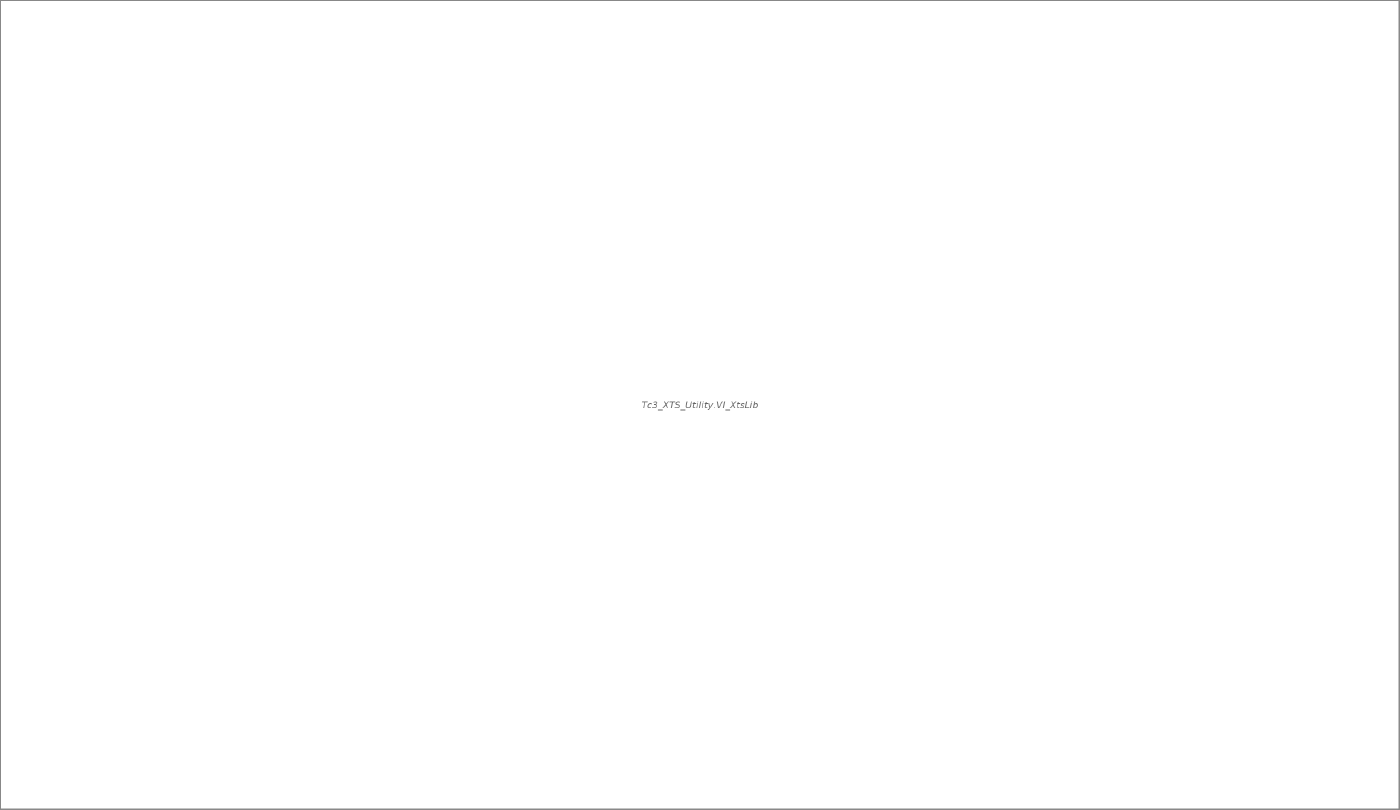
VISUALIZATION PageXtsDiagnostic  // 1520x880
    Frame (0,0 1520x880)
        shows Tc3_XTS_Utility.VI_XtsLib()
END_VISUALIZATION

// ---- VISUs/Recipes/SingleRecipesParameterTypeBool.TcVIS
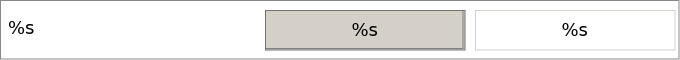
VISUALIZATION SingleRecipesParameterTypeBool  // 680x60
VAR_IN_OUT
	stRecipeParameter : ST_VisuCtrlRecipeParameter;
END_VAR
    Textfield (475,10 200x40), "%s", text variable: stRecipeParameter.sFileValue
    Textfield (5,8 250x40), "%s", text variable: stRecipeParameter.sName
    Button (265,10 200x40), "%s", text variable: stRecipeParameter.sName
        toggle stRecipeParameter.bValue
END_VISUALIZATION

// ---- VISUs/Recipes/SingleRecipesParameterTypeInteger.TcVIS
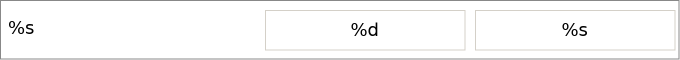
VISUALIZATION SingleRecipesParameterTypeInteger  // 680x60
VAR_IN_OUT
	stRecipeParameter : ST_VisuCtrlRecipeParameter;
END_VAR
    Textfield (265,10 200x40), "%d", text variable: stRecipeParameter.iValue
        OnMouseClick: write the text variable via VisuDialogs.Numpad
    Textfield (475,10 200x40), "%s", text variable: stRecipeParameter.sFileValue
    Textfield (5,8 250x40), "%s", text variable: stRecipeParameter.sName
END_VISUALIZATION

// ---- VISUs/Recipes/SingleRecipesParameterTypeReal.TcVIS
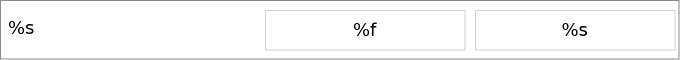
VISUALIZATION SingleRecipesParameterTypeReal  // 680x60
VAR_IN_OUT
	stRecipeParameter : ST_VisuCtrlRecipeParameter;
END_VAR
    Textfield (265,10 200x40), "%f", text variable: stRecipeParameter.rValue
        OnMouseClick: write the text variable via VisuDialogs.Numpad
    Textfield (475,10 200x40), "%s", text variable: stRecipeParameter.sFileValue
    Textfield (5,8 250x40), "%s", text variable: stRecipeParameter.sName
END_VISUALIZATION

// ---- VISUs/Recipes/SingleRecipesParameterTypeString.TcVIS
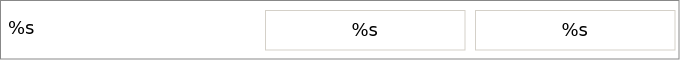
VISUALIZATION SingleRecipesParameterTypeString  // 680x60
VAR_IN_OUT
	stRecipeParameter : ST_VisuCtrlRecipeParameter;
END_VAR
    Textfield (265,10 200x40), "%s", text variable: stRecipeParameter.sValue
        OnMouseClick: write the text variable via VisuDialogs.Keypad
    Textfield (475,10 200x40), "%s", text variable: stRecipeParameter.sFileValue
    Textfield (5,8 250x40), "%s", text variable: stRecipeParameter.sName
END_VISUALIZATION

// ---- VISUs/Recipes/Text Lists/TL_RecipesManagerReturns.TcTLO
TEXTLIST TL_RecipesManagerReturns
  0 = '-'
  10 = 'Operation failed'
  20 = 'Incorrect parameters'
  30 = 'The data server object is not initialized'
  40 = 'The data server does not implement'
  50 = 'Not all variables of a recipe definition can be written via the data server'
  60 = 'The recipe definition has no free memory to create a new recipe'
  70 = 'The recipe file was not found'
  80 = 'The contents of the recipe file do not match the current recipe'
  90 = 'The storage procedure failed'
  100 = 'The recipe does not exist'
  110 = 'The recipe definition does not exist'
  120 = 'The recipe already exists in the recipe definition'
  130 = 'The global recipe manager has not been created'
  140 = 'The recipe definition contains more variables than the recipe file'
  150 = 'The recipe manager was blocked during the online change'
  160 = 'Source exhausted'
  170 = 'Target exhausted'
  180 = 'Source illegal'
   = ''
END_TEXTLIST

// ---- VISUs/Recipes/Text Lists/TL_RecipesManagerStatus.TcTLO
TEXTLIST TL_RecipesManagerStatus
  0 = 'Idle'
  10 = 'Initialization'
  20 = 'Create'
  30 = 'Load'
  40 = 'Read'
  50 = 'Reload'
  60 = 'Backup'
  70 = 'Restore'
  -10 = 'Abort'
   = ''
END_TEXTLIST
